{attribute addProperty BoxType "EL1502-0000-0018"}
{attribute addProperty Id "Enable_output_functionsBIT10.1251Set_outputBIT10.1252Set_counterBIT10.1253Inhibit_counterBIT10.1254"}
{attribute addProperty CRC "512402565"}
{attribute addProperty SizeInBites "16"}
{attribute addProperty SizeInBytes "2"}
TYPE Control_1E8AA485 :
STRUCT
	{attribute addProperty Name "Enable_output_functions"}
	Enable_output_functions : BIT;
	{attribute addProperty Name "Set_output"}
	Set_output : BIT;
	{attribute addProperty Name "Set_counter"}
	Set_counter : BIT;
	{attribute addProperty Name "Inhibit_counter"}
	Inhibit_counter : BIT;
	{attribute 'hide'}
	reserve_1_BIT_0 : BIT;
	{attribute 'hide'}
	reserve_1_BIT_1 : BIT;
	{attribute 'hide'}
	reserve_1_BIT_2 : BIT;
	{attribute 'hide'}
	reserve_1_BIT_3 : BIT;
	{attribute 'hide'}
	reserve_1_BIT_4 : BIT;
	{attribute 'hide'}
	reserve_1_BIT_5 : BIT;
	{attribute 'hide'}
	reserve_1_BIT_6 : BIT;
	{attribute 'hide'}
	reserve_1_BIT_7 : BIT;
	{attribute 'hide'}
	reserve_1_BIT_8 : BIT;
	{attribute 'hide'}
	reserve_1_BIT_9 : BIT;
	{attribute 'hide'}
	reserve_1_BIT_10 : BIT;
	{attribute 'hide'}
	reserve_1_BIT_11 : BIT;
END_STRUCT
END_TYPE

(* stored: Version 1.2.0.0, ProductVersion 3.1.4024.9
   DUT Control_1E8AA485: Id {f2743aae-8803-45d6-9f72-d519da3713f5} *)
